FUNCTION normalizeAngle : LREAL
VAR_INPUT
	angle: LREAL;
	upperBound:LREAL := pi;
	lowerBound:LREAL := -pi;
END_VAR
VAR
END_VAR

IF angle > upperBound THEN
	normalizeAngle := angle - 2*pi;
ELSIF angle < lowerBound THEN
	normalizeAngle := angle + 2*pi;
ELSE
	normalizeAngle := angle;
END_IF

END_FUNCTION

(* stored: Version 1.1.0.1, ProductVersion 3.1.4024.11
   POU normalizeAngle: Id {dcf0afd6-8216-4551-a2e7-b170fbea7d1e}, SpecialFunc None *)
